FUNCTION_BLOCK BaseDamper
VAR_INPUT
	Open: REFERENCE TO BOOL;
	IsOpen: REFERENCE TO BOOL;
	IsClosed: REFERENCE TO BOOL;
END_VAR
VAR_OUTPUT
END_VAR
VAR
END_VAR

END_FUNCTION_BLOCK

(* stored: Version 1.1.0.1, ProductVersion 3.1.4024.3
   POU BaseDamper: Id {e494647b-56ae-454d-af7e-56fa3303edfc}, SpecialFunc None *)
